TYPE EcCoeSdo_Output_typ :
	STRUCT
		Read		: EcCoeSdo_Status_typ ;
		Write		: EcCoeSdo_Status_typ ;
	END_STRUCT
END_TYPE

(* stored: Version 1.1.0.1, ProductVersion 3.1.4024.3
   DUT EcCoeSdo_Output_typ: Id {88d06eae-72d8-050c-322a-6d97cb093688} *)
